// TIA Portal V21 export
TYPE "udt_ABC"
   STRUCT
      "A" : Bool;
      "B" : Bool;
      C : Bool;
   END_STRUCT;
END_TYPE
